{attribute 'Tc2GvlVarNames'}
VAR_GLOBAL

(*METS TPD - PAOL (CML) *)
(*TERMINAL 546KF1 - EK1100 ******************************************************)

(*TERMINAL 547KF2 - EL4002 ******************************************************)

	qn547KF1_1_LightingIntensity						AT %Q* : INT; (*547KF1_1*)
	qn547KF1_2_Spare								AT %Q* : INT; (*547KF1_2*)

(*TERMINAL 560KF1 - EL1008 ******************************************************)
	ib560KF1_1_PrePackAggregationCameraRigTrigger		AT %I* : BOOL; (* 560KF1_1 *)
	ib560KF1_5_PackAggregationCamera1Trigger			AT %I* : BOOL; (* 560KF1_5 *)
	ib560KF1_2_PackAggregationCamera2Trigger			AT %I* : BOOL; (* 560KF1_2 *)
	ib560KF1_6_PackAggregationCamera3Trigger			AT %I* : BOOL; (* 560KF1_6 *)
	ib560KF1_3_PreMachineBuildBack					AT %I* : BOOL; (* 560KF1_3 *)
	ib560KF1_7_TPDExitBlock							AT %I* : BOOL; (* 560KF1_7 *)
	ib560KF1_4_ConveyorIndexContact					AT %I* : BOOL; (* 560KF1_4 *)		(*not used on C922 and C925 *)
	ib560KF1_8_PackIsolatorDrive						AT %I* : BOOL; (* 560KF1_8 *)

(*TERMINAL 5480KF1 - EL2008 ******************************************************)
	qb580KF1_1_PackAggregationCamera1Enable			AT %Q* : BOOL; (* 580KF1_1 *)
	qb580KF1_5_PackAggregationCamera2Enable			AT %Q* : BOOL; (* 580KF1_5 *)
	qb580KF1_2_PackAggregationCamera3Enable			AT %Q* : BOOL; (* 580KF1_2 *)
	qb580KF1_6_PackAggregationCamera1Power			AT %Q* : BOOL; (* 580KF1_6 *)
	qb580KF1_3_PackAggregationCamera2Power			AT %Q* : BOOL; (* 580KF1_3 *)
	qb580KF1_7_PackAggregationCamera3Power			AT %Q* : BOOL; (* 580KF1_7 *)
	qb580KF1_4_Spare								AT %Q* : BOOL; (* 580KF1_4 *)
	qb580KF1_8_PackCamerasLenseAir					AT %Q* : BOOL; (* 580KF1_8 *)

END_VAR

(* stored: Version 1.1.0.1, ProductVersion 3.1.4024.15
   GVL IOVariablesPAOL_CML: Id {ad609d10-efa7-475b-8826-2cd3b6720411} *)
